//SimpleTrajectory:
//implements a simple trajectory which takes a waypoint list od max 100 poses. The points are outputted one by one as reference pose with no further modifications.
//The trajectory switches to the next pose if the x-y-distance d between  'currentPose' and the current reference 'referencePose[WPLidx]'
//is within a tolerance 'tol' to the current . TODO: modify d such it represents a x-y-theta distance. 
//waypoint. If all three coordinates of the waypoint are set to -1 the trajectory marks itself
//as finished.
FUNCTION_BLOCK SimpleTrajectory
VAR_INPUT
	currentPose			: RobotPoseSimple;
END_VAR
VAR_OUTPUT
	finished			: BOOL 				:= FALSE;
	referencePose		: RobotPoseSimple;
	WPLidx 				: INT 				:= 0;
END_VAR
VAR
	wayPointList		: ARRAY [0..100] OF RobotPoseSimple;
	d: LREAL  := 0;
	tol: LREAL := 10; 
END_VAR

//calculte current distance from reference point
d := SQRT(EXPT(currentPose.x - wayPointList[WPLidx].x, 2) + EXPT(currentPose.y - wayPointList[WPLidx].y,2));

IF d < tol AND NOT finished THEN
	WPLidx := WPLidx +1;
END_IF

IF wayPointList[WPLidx].x = -1 AND wayPointList[WPLidx].y = -1 AND wayPointList[WPLidx].theta = -1 THEN
	finished := TRUE;
END_IF

referencePose := wayPointList[WPLidx];

METHOD getReferencePose : RobotPoseSimple
VAR_INPUT
END_VAR
END_METHOD

METHOD setRobotPose : RobotPoseSimple
VAR_INPUT
	newPose: RobotPoseSimple;
END_VAR
setRobotPose := newPose;
END_METHOD

METHOD setWaypointList : ARRAY [0..100] OF RobotPoseSimple
VAR_INPUT
	newWayPointList	: ARRAY [0..100]  OF RobotPoseSimple;
END_VAR
WPLidx 			:= 0; 						//reset
finished 		:= FALSE;
wayPointList 	:= newWayPointList;
END_METHOD

END_FUNCTION_BLOCK

(* stored: Version 1.1.0.1, ProductVersion 3.1.4024.11
   POU SimpleTrajectory: Id {17c71041-eda0-416f-945f-5d35424906cd}, SpecialFunc None
   Method getReferencePose: Id {5ec1042d-abfb-4a75-8fd5-89022b6f0e89}
   Method setRobotPose: Id {612c742a-1fe7-4003-9836-d6bbc0467a35}
   Method setWaypointList: Id {e85e045f-80a3-4da6-9e39-79af30febaa9} *)
